TYPE T_AVL_Node : ST_AVL_NODE; END_TYPE

(* stored: Version 1.1.0.1, ProductVersion 3.1.4024.4
   DUT T_AVL_Node: Id {db32b49b-11ed-0512-249d-11105767d55e} *)
